# EPICS substitutions: ioc-tmo-output-couplerApp/Db/tmo-output-coupler.substitutions
file "db/tmo-output-coupler.db" {
    { P = "ioc-tmo-output-coupler" }
}
